## Short summary
This property returns an ``ICycleError`` interface fluently to provide error handling methods.

.. <legal notes>

legal notes
=================
| SPDX-FileCopyrightText: © 2024 ekvip automation GmbH <info@ekvip.de>
| SPDX-License-Identifier: Apache-2.0
| For details check: Apache-2.0_

.. _Apache-2.0: https://www.apache.org/licenses/LICENSE-2.0

.. </legal notes>

*)
PROPERTY errors : CNM_CycleManagerInterfaces.ICycleError
GET
errors := THIS^;
END_GET
END_PROPERTY

(*

## Short summary
This method evaluates an execution state to calculate the next step.

.. <legal notes>

legal notes
=================
| SPDX-FileCopyrightText: © 2024 ekvip automation GmbH <info@ekvip.de>
| SPDX-License-Identifier: Apache-2.0
| For details check: Apache-2.0_

.. _Apache-2.0: https://www.apache.org/licenses/LICENSE-2.0

.. </legal notes>

*)
METHOD evaluate
VAR_INPUT
	(* the state which is to be evaluated *)
	state	:CNM_ReturnTypes.SingleExecutionState;
	(* step to proceed with in case of error *)
	errorStep	:DINT := CNM_ReturnTypes.DefaultSteps.STEP.ERROR;
END_VAR
THIS^.registeredEval := TRUE;

RETURN ( 	
		THIS^.wasError 
	OR_ELSE 
		(THIS^.state <> CNM_ReturnTypes.SingleExecutionState.BUSY)
	OR_ELSE
		NOT THIS^.executeStep
);

CASE state OF
CNM_ReturnTypes.SingleExecutionState.ERROR, CNM_ReturnTypes.SingleExecutionState.ABORTED:
	THIS^.wasError := TRUE;
	THIS^.wasSuccess := FALSE;
	IF ((errorStep <> CNM_ReturnTypes.DefaultSteps.STEP.ERROR) 
		AND_THEN (errorStep <> THIS^.currentErrorStep)
	) THEN
		THIS^.currentErrorStep := errorStep;
	END_IF
CNM_ReturnTypes.SingleExecutionState.BUSY:
	THIS^.wasNotSuccess := TRUE;
	IF(NOT THIS^.wasError)THEN
		THIS^.wasSuccess := FALSE;
	END_IF
CNM_ReturnTypes.SingleExecutionState.SUCCESS:
	IF(NOT THIS^.wasError AND NOT THIS^.wasNotSuccess)THEN
		THIS^.wasSuccess := TRUE;	
	END_IF
CNM_ReturnTypes.SingleExecutionState.IDLE, CNM_ReturnTypes.SingleExecutionState.PAUSED:
	THIS^.wasNotSuccess := TRUE;
	IF(NOT THIS^.wasError)THEN
		THIS^.wasSuccess := FALSE;
	END_IF
END_CASE
END_METHOD

(*

## Short summary
This method performs the given command and evaluates the return value.
The command will be called with execute := FALSE in the first cylce and with execute := TRUE in all following

.. <legal notes>

legal notes
=================
| SPDX-FileCopyrightText: © 2024 ekvip automation GmbH <info@ekvip.de>
| SPDX-License-Identifier: Apache-2.0
| For details check: Apache-2.0_

.. _Apache-2.0: https://www.apache.org/licenses/LICENSE-2.0

.. </legal notes>

*)
METHOD executeCommand
VAR_INPUT
	(* command to execute *)
	command :CNM_CommandInterfaces.ICommand;
	(* step to proceed with in case of error *)
	errorStep :DINT := CNM_ReturnTypes.DefaultSteps.STEP.ERROR;
END_VAR
THIS^.registeredCommand := TRUE;

IF(THIS^.isObjectNull(command))THEN
	THIS^.evaluate(CNM_ReturnTypes.SingleExecutionState.ERROR, errorStep);	
ELSE
	THIS^.evaluate(command.executeCommand(THIS^.executeStep), errorStep);	
END_IF
END_METHOD

(*

## Short summary
This property returns the execute flag for the current step, 
which is FALSE in the first cycle of each step and TRUE after.

.. <legal notes>

legal notes
=================
| SPDX-FileCopyrightText: © 2024 ekvip automation GmbH <info@ekvip.de>
| SPDX-License-Identifier: Apache-2.0
| For details check: Apache-2.0_

.. _Apache-2.0: https://www.apache.org/licenses/LICENSE-2.0

.. </legal notes>

*)
PROPERTY executeStep :BOOL
GET
executeStep := THIS^.externalExecute;
END_GET
END_PROPERTY

METHOD PROTECTED getStateFromStep : CNM_ReturnTypes.SingleExecutionState
VAR_INPUT
	step :DINT;
END_VAR
CASE step OF
STEP_ABORT:
	getStateFromStep := CNM_ReturnTypes.SingleExecutionState.ABORTED;
STEP_ERROR:
	getStateFromStep := CNM_ReturnTypes.SingleExecutionState.ERROR;
STEP_PAUSE:
	getStateFromStep := CNM_ReturnTypes.SingleExecutionState.PAUSED;
STEP_SUCCESS:
	getStateFromStep := CNM_ReturnTypes.SingleExecutionState.SUCCESS;
STEP_IDLE:
	;
STEP_INIT:
	getStateFromStep := CNM_ReturnTypes.SingleExecutionState.BUSY;
ELSE
	//sequence is running
	getStateFromStep := CNM_ReturnTypes.SingleExecutionState.BUSY;
END_CASE
END_METHOD

(*

## Short summary
This method throws an alarm and waits for it to be confirmed. 
When the alarm was confirmed the cyclemanager will proceed to next configured step.
If the current step is the result of an evaulated error state and the input 'resumeWithLastStep' is set to true, the cyclemanager will proceed to the last step.
..warning:  The 'resumeWithLastStep' flag will be ignored if the last step was successful.

.. <legal notes>

legal notes
=================
| SPDX-FileCopyrightText: © 2024 ekvip automation GmbH <info@ekvip.de>
| SPDX-License-Identifier: Apache-2.0
| For details check: Apache-2.0_

.. _Apache-2.0: https://www.apache.org/licenses/LICENSE-2.0

.. </legal notes>

*)

METHOD handle
VAR_INPUT
	(* the alarm event that should be thrown *)
	alarm :CNM_MessageInterfaces.IAlarm;
	(* if this flag is set AND we got to the current step because of an ERROR state, then the cyclemanager will automatically will go back to the last step *)
	resumeWithLastStep :BOOL := TRUE;
END_VAR
IF(NOT THIS^.executeStep)THEN
	alarm.throw();
ELSIF(NOT alarm.isPending)THEN
	IF(resumeWithLastStep AND_THEN THIS^.gotHereByError)THEN
		THIS^.acknowledge();
	ELSE
		THIS^.evaluate(state := CNM_ReturnTypes.SingleExecutionState.SUCCESS);
	END_IF
END_IF
END_METHOD

(*

## Short summary
This method handles the resume function of the cycle manager.
Should be called befor all other handles.

.. <legal notes>

legal notes
=================
| SPDX-FileCopyrightText: © 2024 ekvip automation GmbH <info@ekvip.de>
| SPDX-License-Identifier: Apache-2.0
| For details check: Apache-2.0_

.. _Apache-2.0: https://www.apache.org/licenses/LICENSE-2.0

.. </legal notes>

*)
METHOD PROTECTED handleCycleManagerError
VAR_INPUT
	(*if true, will acknowledge error and return to previous step*)
	resume :BOOL;
END_VAR
IF(resume)THEN
	THIS^.acknowledge();
END_IF
END_METHOD

(*

## Short summary
This method handles the execution of the cycle manager.
Should be the first thing to do at the start of each cycle.

.. <legal notes>

legal notes
=================
| SPDX-FileCopyrightText: © 2024 ekvip automation GmbH <info@ekvip.de>
| SPDX-License-Identifier: Apache-2.0
| For details check: Apache-2.0_

.. _Apache-2.0: https://www.apache.org/licenses/LICENSE-2.0

.. </legal notes>

*)
METHOD PROTECTED handleCycleManagerExecute : BOOL
VAR_INPUT
	(*control bit to start or abort the cycle manager*)
	execute :BOOL;
END_VAR
IF(THIS^.lastExecute <> execute)THEN
	IF(execute)THEN
		//first cylce / init
		THIS^.currentState := CNM_ReturnTypes.SingleExecutionState.BUSY;
		THIS^.step.next := STEP_INIT;
		THIS^.firstCycle := TRUE;
	ELSE		
		//falling execute / reset
		IF(THIS^.currentState = CNM_ReturnTypes.SingleExecutionState.BUSY OR THIS^.currentState = CNM_ReturnTypes.SingleExecutionState.PAUSED)THEN
			THIS^.currentState := CNM_ReturnTypes.SingleExecutionState.ABORTED;
			THIS^.currentStep := STEP_ABORT;
		ELSE
			THIS^.currentStep := STEP_IDLE;	
			THIS^.step.next := STEP_IDLE;	
			THIS^.lastStep := STEP_IDLE;			
		END_IF
		THIS^.externalExecute := FALSE;
	END_IF
ELSIF(THIS^.currentStep = STEP_ABORT)THEN
	//only one cycle in ABORT Step
	THIS^.currentStep := STEP_IDLE;
END_IF

THIS^.lastExecute := execute;

handleCycleManagerExecute := execute;
END_METHOD

(*

## Short summary
This method handles the pausing of the cycle manager. 
Should be handled before updating.

.. <legal notes>

legal notes
=================
| SPDX-FileCopyrightText: © 2024 ekvip automation GmbH <info@ekvip.de>
| SPDX-License-Identifier: Apache-2.0
| For details check: Apache-2.0_

.. _Apache-2.0: https://www.apache.org/licenses/LICENSE-2.0

.. </legal notes>

*)
METHOD PROTECTED handleCycleManagerPause
VAR_INPUT
	(*if true and Pausing Enabled and busy will proceed with PAUSE*)
	pause :BOOL;
END_VAR
IF(NOT pause AND_THEN THIS^.currentState = CNM_ReturnTypes.SingleExecutionState.PAUSED)THEN
	THIS^.currentStep := THIS^.lastStepBeforePause;
END_IF

RETURN (NOT THIS^.currentPauseEnabled);

IF(
	pause 
	AND_THEN (NOT THIS^.wasError) 
	AND_THEN (THIS^.currentState = CNM_ReturnTypes.SingleExecutionState.BUSY)
)THEN
	THIS^.lastStepBeforePause := THIS^.currentStep;
	THIS^.currentStep := STEP_PAUSE;
END_IF
END_METHOD

(*

## Short summary
This method handles the timeout of the current step.
Call at any point each cycle.
.. <legal notes>

legal notes
=================
| SPDX-FileCopyrightText: © 2024 ekvip automation GmbH <info@ekvip.de>
| SPDX-License-Identifier: Apache-2.0
| For details check: Apache-2.0_

.. _Apache-2.0: https://www.apache.org/licenses/LICENSE-2.0

.. </legal notes>

*)
METHOD PROTECTED handleCycleManagerTimeout : BOOL
VAR_INPUT
	(* must be TRUE if stepping is enabled to proceed steps automatically *)
	step :BOOL;
END_VAR
IF ((THIS^.currentState = CNM_ReturnTypes.SingleExecutionState.BUSY) AND (THIS^.currentTimeout > T#0S)) THEN
	THIS^.timeoutTimer(
		IN := (
			(NOT THIS^.currentSteppingEnabled) 
			OR 
			(NOT step)
		), 
		PT := THIS^.currentTimeout,
		Q => THIS^.wasTimeoutError
	);
END_IF
END_METHOD

(*

## Short summary
This method handles the step change, call early in handling.

.. <legal notes>

legal notes
=================
| SPDX-FileCopyrightText: © 2024 ekvip automation GmbH <info@ekvip.de>
| SPDX-License-Identifier: Apache-2.0
| For details check: Apache-2.0_

.. _Apache-2.0: https://www.apache.org/licenses/LICENSE-2.0

.. </legal notes>

*)
METHOD PROTECTED handleStepChange
VAR_INPUT
	(* must be TRUE if stepping is enabled to proceed steps automatically *)
	step :BOOL := TRUE;
	(*used for StopRequest evaluation if configured*)
	stopRequest :BOOL := FALSE;
END_VAR
IF THIS^.wasError THEN
    THIS^.step.next := THIS^.currentErrorStep;
    THIS^.initializeNewStep(TRUE);

ELSIF THIS^.wasTimeoutError THEN
    THIS^.step.next := THIS^.currentTimeoutStep;
    THIS^.initializeNewStep(TRUE);

ELSIF stopRequest AND (
        (THIS^.wasSuccess AND NOT THIS^.wasNotSuccess AND (THIS^.executeStep OR NOT THIS^.isAnyActionRegistered)
            AND THIS^.currentStopRequestMode = CNM_CycleManagerInterfaces.StepStopRequestMode.AFTER_SUCCESSFUL_STEP)
     OR (THIS^.wasNotSuccess AND (THIS^.executeStep OR NOT THIS^.isAnyActionRegistered)
            AND THIS^.currentStopRequestMode = CNM_CycleManagerInterfaces.StepStopRequestMode.ON_BUSY)
     OR (THIS^.currentStopRequestMode = CNM_CycleManagerInterfaces.StepStopRequestMode.IMMEDIATE)
) THEN
    THIS^.step.next := STEP_SUCCESS;
    THIS^.initializeNewStep();

ELSIF THIS^.wasSuccess
	AND NOT THIS^.wasNotSuccess 
	AND (THIS^.executeStep OR NOT THIS^.isAnyActionRegistered)
    AND (NOT THIS^.currentSteppingEnabled OR step) 
THEN
    THIS^.initializeNewStep();
END_IF
END_METHOD

METHOD PRIVATE initializeNewStep
VAR_INPUT
	errorStep :BOOL := FALSE;
END_VAR
THIS^.gotHereByError := errorStep;
THIS^.firstCycle := TRUE;
END_METHOD

(*

## Short summary
This boolean is true when at least one of these actions are registered:
- executeCommand
- evaluate
- leave

The setter can be used to clear all the registered actions at once. 

.. <legal notes>

legal notes
=================
| SPDX-FileCopyrightText: © 2025 ekvip automation GmbH <info@ekvip.de>
| SPDX-License-Identifier: Apache-2.0
| For details check: Apache-2.0_

.. _Apache-2.0: https://www.apache.org/licenses/LICENSE-2.0

.. </legal notes>

*)

PROPERTY PROTECTED isAnyActionRegistered : BOOL
GET
isAnyActionRegistered := THIS^.registeredCommand OR THIS^.registeredLeave OR THIS^.registeredEval;
END_GET
SET
RETURN(isAnyActionRegistered); //dont set all the flags to true at once
THIS^.registeredCommand := 
THIS^.registeredEval := 
THIS^.registeredLeave := isAnyActionRegistered; // only if isAnyActionRegistered is set to false
END_SET
END_PROPERTY

(*

## Short summary
This property returns TRUE if the step was reached by evaluating an error.

.. <legal notes>

legal notes
=================
| SPDX-FileCopyrightText: © 2024 ekvip automation GmbH <info@ekvip.de>
| SPDX-License-Identifier: Apache-2.0
| For details check: Apache-2.0_

.. _Apache-2.0: https://www.apache.org/licenses/LICENSE-2.0

.. </legal notes>

*)
{attribute 'hide'}
PROPERTY isInErrorStep :BOOL
GET
isInErrorStep := THIS^.gotHereByError;
END_GET
END_PROPERTY

(*

## Short summary
This property returns the last step of the cycle manager, useful for error steps.

.. <legal notes>

legal notes
=================
| SPDX-FileCopyrightText: © 2024 ekvip automation GmbH <info@ekvip.de>
| SPDX-License-Identifier: Apache-2.0
| For details check: Apache-2.0_

.. _Apache-2.0: https://www.apache.org/licenses/LICENSE-2.0

.. </legal notes>

### Example
```
TIMEOUT_STEP_FOR_RETRY:
	cM.steps.next := cM.steps.last-1;
	cM.waitFor(ACK);

*)
{attribute 'hide'}
PROPERTY last : DINT
GET
last := SEL(THIS^.currentStep = STEP_PAUSE, THIS^.lastStep, THIS^.lastStepBeforePause);
END_GET
SET // PROTECTED
THIS^.lastStep := last;
END_SET
END_PROPERTY

(*

## Short summary
This method performs the given invoke only in the last cycle of the current step.

.. <legal notes>

legal notes
=================
| SPDX-FileCopyrightText: © 2024 ekvip automation GmbH <info@ekvip.de>
| SPDX-License-Identifier: Apache-2.0
| For details check: Apache-2.0_

.. _Apache-2.0: https://www.apache.org/licenses/LICENSE-2.0

.. </legal notes>

*)
METHOD leave
VAR_INPUT
	(* command to execute *)
	invoke	:CNM_CommandInterfaces.ISingleAttempt;
	(* step to proceed with in case of error *)
	errorStep	:DINT := CNM_ReturnTypes.DefaultSteps.STEP.ERROR; 
	(* whether the invoke should be called even if there was an error in the current step *)
	forceOnError	:BOOL := FALSE;
END_VAR
THIS^.registeredLeave := TRUE;

RETURN ((
			((NOT wasSuccess) OR_ELSE THIS^.wasNotSuccess) 
		AND 
			NOT(forceOnError AND THIS^.wasError)
		) 
	OR 
		THIS^.state <> CNM_ReturnTypes.SingleExecutionState.BUSY
);

IF(THIS^.isObjectNull(invoke) OR_ELSE invoke.invoke() <> CNM_ReturnTypes.SingleExecutionResult.SUCCESS)THEN
	THIS^.evaluate(CNM_ReturnTypes.SingleExecutionState.ERROR, errorStep);	
END_IF
END_METHOD

(*

## Short summary
This property sets the next step of the cycle manager.

.. <legal notes>

legal notes
=================
| SPDX-FileCopyrightText: © 2024 ekvip automation GmbH <info@ekvip.de>
| SPDX-License-Identifier: Apache-2.0
| For details check: Apache-2.0_

.. _Apache-2.0: https://www.apache.org/licenses/LICENSE-2.0

.. </legal notes>

### Example
```
MY_STEP:
	cyclemanager.steps.next := SUCCESS_STEP;
	cyclemanager.executeCommand(finalizeProcess);
	
*)
{attribute 'hide'}
PROPERTY next : DINT
GET
next := SEL(THIS^.nextStepSpecifiedByUser, THIS^.currentStep + THIS^.currentStepWidth, THIS^.nextStep);
END_GET
SET
THIS^.nextStep := next;
THIS^.nextStepSpecifiedByUser := TRUE;
END_SET
END_PROPERTY

(*

## Short summary
This method changes the current step in the cycle manager to the next in order (current + stepWidth) .
If any evaluate or other call is still busy it will ignore them and change to the next step.

.. <legal notes>

legal notes
=================
| SPDX-FileCopyrightText: © 2024 ekvip automation GmbH <info@ekvip.de>
| SPDX-License-Identifier: Apache-2.0
| For details check: Apache-2.0_

.. _Apache-2.0: https://www.apache.org/licenses/LICENSE-2.0

.. </legal notes>

*)
METHOD proceed
RETURN (THIS^.state = CNM_ReturnTypes.SingleExecutionState.SUCCESS);

THIS^.wasNotSuccess := FALSE;
THIS^.wasSuccess := TRUE;
THIS^.isAnyActionRegistered := FALSE;
END_METHOD

(*

## Short summary
This method changes the current step in the cycle manager to the given step.
If any evaluate or other call is still busy it will ignore them and move to the next step.

.. <legal notes>

legal notes
=================
| SPDX-FileCopyrightText: © 2024 ekvip automation GmbH <info@ekvip.de>
| SPDX-License-Identifier: Apache-2.0
| For details check: Apache-2.0_

.. _Apache-2.0: https://www.apache.org/licenses/LICENSE-2.0

.. </legal notes>

*)
METHOD proceedWith
VAR_INPUT
	(* step to move to *)
	step	:DINT;
END_VAR
RETURN (THIS^.state = CNM_ReturnTypes.SingleExecutionState.SUCCESS);

THIS^.step.next := step;
THIS^.proceed();
END_METHOD

METHOD PROTECTED resetCurrentStepParametersToDefaults
VAR_INPUT
END_VAR
THIS^.currentErrorStep := THIS^.defaultErrorStep;
THIS^.currentPauseEnabled := THIS^.defaultPauseEnabled;
THIS^.currentSteppingEnabled := THIS^.defaultSteppingEnabled;
THIS^.currentStepWidth := THIS^.defaultStepWidth;
THIS^.currentStopRequestMode := THIS^.defaultStopRequestMode;
THIS^.currentTimeoutStep := THIS^.defaultTimeoutStep;
THIS^.currentTimeout := THIS^.defaultTimeout;
END_METHOD

METHOD PROTECTED resetInternalVariables
THIS^.registeredCommand := FALSE;
THIS^.registeredEnter := FALSE;
THIS^.registeredEval := FALSE;
THIS^.registeredLeave := FALSE;	
THIS^.wasError := FALSE;
THIS^.wasTimeoutError := FALSE;
THIS^.wasNotSuccess := FALSE;
THIS^.wasSuccess := FALSE;
THIS^.firstCycle := FALSE;
THIS^.nextStepSpecifiedByUser := FALSE;
END_METHOD

(*

## Short summary
This property returns the current state of the cycle manager according to its step.

.. <legal notes>

legal notes
=================
| SPDX-FileCopyrightText: © 2024 ekvip automation GmbH <info@ekvip.de>
| SPDX-License-Identifier: Apache-2.0
| For details check: Apache-2.0_

.. _Apache-2.0: https://www.apache.org/licenses/LICENSE-2.0

.. </legal notes>

*)
PROPERTY state : CNM_ReturnTypes.SingleExecutionState
GET
VAR CONSTANT
	WAITING : DINT := 42;
END_VAR
IF(
	NOT THIS^.sequenceRequireSuccessStep
	AND_THEN NOT THIS^.wasError 
	AND_THEN wasSuccess 
	AND_THEN (THIS^.executeStep OR NOT(THIS^.registeredEval OR THIS^.registeredCommand OR THIS^.registeredLeave))
	AND_THEN THIS^.step.next = STEP_SUCCESS
)THEN
	//this allows the cycle manager to return SUCCESS one cycle earlier, saving many cycles in nested use
	THIS^.currentState := CNM_ReturnTypes.SingleExecutionState.SUCCESS;
END_IF

state := THIS^.currentState;
END_GET
SET // PROTECTED
THIS^.currentState := state;
END_SET
END_PROPERTY

(*

## Short summary
This property returns the current, next and last step of the cycle manager via fluent interface with the ``ICylceSteps`` interfaces

.. <legal notes>

legal notes
=================
| SPDX-FileCopyrightText: © 2024 ekvip automation GmbH <info@ekvip.de>
| SPDX-License-Identifier: Apache-2.0
| For details check: Apache-2.0_

.. _Apache-2.0: https://www.apache.org/licenses/LICENSE-2.0

.. </legal notes>

*)
PROPERTY step : CNM_CycleManagerInterfaces.ICycleSteps
GET
step := THIS^;
END_GET
END_PROPERTY

(*

## Short summary
This method handles all updates of the cycle manager.
Should be called first each cycle befor evaluating the steps and only once per cycle!

.. <legal notes>

legal notes
=================
| SPDX-FileCopyrightText: © 2024 ekvip automation GmbH <info@ekvip.de>
| SPDX-License-Identifier: Apache-2.0
| For details check: Apache-2.0_

.. _Apache-2.0: https://www.apache.org/licenses/LICENSE-2.0

.. </legal notes>

*)
METHOD update
VAR_INPUT
	(*control bit to start or abort the cycle manager*)
	execute :BOOL;
	(*used for StopRequest evaluation if configured*)
	stopRequest :BOOL := FALSE;
	(*if true and Pausing Enabled and busy will proceed with PAUSE*)
	pause :BOOL := FALSE;
	(*if true, will acknowledge error and return to previous step*)
	resume :BOOL := FALSE;
	(* must be TRUE if stepping is enabled to proceed steps automatically *)
	stepControl :BOOL := TRUE;
END_VAR
RETURN (NOT THIS^.handleCycleManagerExecute(execute));
THIS^.handleCycleManagerError(resume);
THIS^.handleStepChange(stepControl, stopRequest);
THIS^.handleCycleManagerPause(pause);
THIS^.handleCycleManagerTimeout(stepControl);
THIS^.updateCycleManager();
END_METHOD

(*

## Short summary
This method updates the step and state of the cycle manager.
Should be called after all handles each cycle.

.. <legal notes>

legal notes
=================
| SPDX-FileCopyrightText: © 2024 ekvip automation GmbH <info@ekvip.de>
| SPDX-License-Identifier: Apache-2.0
| For details check: Apache-2.0_

.. _Apache-2.0: https://www.apache.org/licenses/LICENSE-2.0

.. </legal notes>

*)
METHOD PROTECTED updateCycleManager
THIS^.externalExecute := NOT THIS^.firstCycle;

IF (THIS^.firstCycle AND_THEN (THIS^.currentStep <> CNM_ReturnTypes.DefaultSteps.STEP.SUCCESS)) THEN
	THIS^.timeoutTimer(IN := FALSE);
	
	THIS^.last := THIS^.currentStep;
	THIS^.currentStep := THIS^.step.next;
	
	THIS^.resetInternalVariables();
	THIS^.resetCurrentStepParametersToDefaults();
END_IF

//Set State for external use
THIS^.state := getStateFromStep(THIS^.currentStep);

THIS^.wasError := FALSE;
THIS^.wasNotSuccess := FALSE;
THIS^.wasSuccess := FALSE;
END_METHOD

(*

## Short summary
This method waits for a boolean signal until the step can be changed. 

.. <legal notes>

legal notes
=================
| SPDX-FileCopyrightText: © 2024 ekvip automation GmbH <info@ekvip.de>
| SPDX-License-Identifier: Apache-2.0
| For details check: Apache-2.0_

.. _Apache-2.0: https://www.apache.org/licenses/LICENSE-2.0

.. </legal notes>

*)
METHOD waitFor
VAR_INPUT
	(* the value to wait for *)
	value	:BOOL;
END_VAR
RETURN (THIS^.state <> CNM_ReturnTypes.SingleExecutionState.BUSY);

THIS^.registeredEval := TRUE;

IF(value)THEN
	IF(NOT wasError)THEN
		THIS^.wasSuccess := TRUE;
	END_IF
ELSE
	THIS^.wasNotSuccess := TRUE;
END_IF
END_METHOD

END_FUNCTION_BLOCK

// ---- CycleManager/classes/SimpleCycleManager.TcPOU
(*

## Short summary
An implementation of the ``ISinlgeExecutionCycleManager`` to provide simple cycle managment for steps in state machines.
The body NEEDS to be called at the start of every cycle (before using the step property) ONLY ONCE.

.. <info>
If used in the same step, the order of method calls should be this:
configurations
enter
executeCommand
evaluate
waitFor
proceed
proceedWith
acknowledge
leave
.. </info>

.. <legal notes>

legal notes
=================
| SPDX-FileCopyrightText: © 2024 ekvip automation GmbH <info@ekvip.de>
| SPDX-License-Identifier: Apache-2.0
| For details check: Apache-2.0_

.. _Apache-2.0: https://www.apache.org/licenses/LICENSE-2.0

.. </legal notes>



*)
FUNCTION_BLOCK SimpleCycleManager EXTENDS AbstractCycleManager
VAR_INPUT
	(*control bit to start or abort the cycle manager*)
	execute :BOOL;
	(*used for StopRequest evaluation if configured*)
	stopRequest :BOOL := FALSE;
	(*if true and Pausing Enabled and busy will proceed with PAUSE*)
	pause :BOOL := FALSE;
	(*if true, will acknowledge error and return to previous step*)
	resume :BOOL := FALSE;
	(* must be TRUE if stepping is enabled to proceed steps automatically *)
	stepControl :BOOL := TRUE;
END_VAR

THIS^.update(
	execute := execute, 
	pause := pause, 
	resume := resume, 
	stepControl := stepControl, 
	stopRequest := stopRequest
);

(*

## Short summary
This abstract property returns the class name of the concrete object, 
which is useful for logging/debugging purpose or to check the class name
for ``__DELETE`` in factories (sometimes it's necessary to do more 
than just to free the memory).

.. <legal notes>

legal notes
=================
| SPDX-FileCopyrightText: © 2022 ekvip automation GmbH <info@ekvip.de>
| SPDX-License-Identifier: Apache-2.0
| For details check: Apache-2.0_

.. _Apache-2.0: https://www.apache.org/licenses/LICENSE-2.0

.. </legal notes>

*)
PROPERTY className : CNM_AbstractObject.ClassName
GET
className := 'CNM_CycleManager.SimpleCycleManager';
END_GET
END_PROPERTY

END_FUNCTION_BLOCK

// ---- Project Information/F_GetCompany.TcPOU
// This function has been automatically generated from the project information.
{attribute 'signature_flag' := '1073741824'}
{attribute 'TcGenerated'}
{attribute 'no-analysis'}
FUNCTION F_GetCompany : WSTRING
VAR_INPUT
	
END_VAR

F_GetCompany := "ekvip automation GmbH";

END_FUNCTION

// ---- Project Information/F_GetTitle.TcPOU
// This function has been automatically generated from the project information.
{attribute 'signature_flag' := '1073741824'}
{attribute 'TcGenerated'}
{attribute 'no-analysis'}
FUNCTION F_GetTitle : WSTRING
VAR_INPUT
	
END_VAR

F_GetTitle := "CNM_CycleManager";

END_FUNCTION

// ---- Project Information/F_GetVersion.TcPOU
// This function has been automatically generated from the project information.
{attribute 'signature_flag' := '1073741824'}
{attribute 'TcGenerated'}
{attribute 'no-analysis'}
FUNCTION F_GetVersion : ST_LibVersion
VAR_INPUT
	
END_VAR

F_GetVersion.iMajor := 0;
F_GetVersion.iMinor := 1;
F_GetVersion.iBuild := 1;
F_GetVersion.iRevision := 0;
F_GetVersion.sVersion := '0.1.1.0';
F_GetVersion.nFlags := 0;

END_FUNCTION
